TYPE ST_Outputs :
STRUCT
	Advance   AT %Q*: BOOL; //Hardware Output Advance Signal
	Retract  AT %Q*: BOOL;  //Hardware Output Retract Signal
END_STRUCT
END_TYPE

(* stored: Version 1.1.0.1, ProductVersion 3.1.4024.12
   DUT ST_Outputs: Id {4d9a78c5-6969-48df-85ea-8b8c83990e3f} *)
